INTERFACE I_Command

METHOD Destroy
VAR_INPUT
END_VAR
END_METHOD

METHOD PUBLIC Execute : BOOL
VAR_INPUT
END_VAR
END_METHOD

PROPERTY PUBLIC isBusy : BOOL
GET
END_GET
END_PROPERTY

PROPERTY isComplete : BOOL
GET
END_GET
END_PROPERTY

END_INTERFACE

(* stored: Version 1.1.0.1, ProductVersion 3.1.4024.9
   Itf I_Command: Id {6f8f5bd7-65cd-4609-92ad-f65effbcf8e5}
   Method Destroy: Id {2a4d2710-f9e8-4537-b240-6283c604cfac}
   Method Execute: Id {8cfea5b9-95ab-4496-9646-77bca8cd2eb8}
   Property isBusy: Id {2ddf0da5-aaa8-4166-8a99-af9430737934}
   Get Get: Id {c90254ea-79a2-45e2-a71a-aa4bf21ad42b}
   Property isComplete: Id {257714a2-9732-4b01-82ab-6b268f7bd803}
   Get Get: Id {037e08c2-cf12-43db-9bad-e0155de62229} *)
